// TwinCAT 3 PLC project CodeAnalysisTcLib
// ProgramVersion: 3.1.4022.7
// project tree:
//   / FB_Math.TcPOU

// ---- FB_Math.TcPOU
FUNCTION_BLOCK FB_Math
VAR_INPUT
END_VAR
VAR_OUTPUT
END_VAR
VAR
END_VAR

METHOD AddTwo : REAL
VAR_INPUT
	Real1 :REAL;
	Real2 :REAL;
END_VAR

AddTwo := Real1 + Real2;
AddTwo := Real1 + Real2;
END_METHOD

END_FUNCTION_BLOCK
